PROGRAM SealedIn
VAR
	Trigger: BOOL;
	Sealed_In_Coil: BOOL;
END_VAR

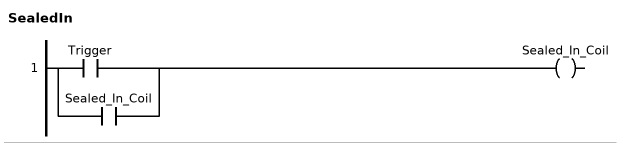
// NETWORK 1
Sealed_In_Coil := Trigger OR Sealed_In_Coil;

END_PROGRAM

(* stored: Version 1.1.0.1, ProductVersion 3.1.4024.10
   POU SealedIn: Id {e70ef259-7506-4c59-83c7-fa25a2ade694}, SpecialFunc None *)
